(* PLC project MQTT, OpenPLC MQTT 1.0, author OpenPLC Lib Writter *)
(* stored: creationDateTime 2023-04-26T04:54:00, modificationDateTime 2023-04-26T04:54:00 *)

(* MQTT_RECEIVE *)
FUNCTION_BLOCK MQTT_RECEIVE
  VAR_INPUT
    RECEIVE : BOOL;  (* RECEIVE *)
    TOPIC : STRING;  (* TOPIC *)
  END_VAR
  VAR_OUTPUT
    RECEIVED : BOOL;  (* RECEIVED *)
    MESSAGE : STRING;  (* MESSAGE *)
  END_VAR

  RECEIVED := 0;
END_FUNCTION_BLOCK

(* MQTT_SEND *)
FUNCTION_BLOCK MQTT_SEND
  VAR_INPUT
    SEND : BOOL;  (* SEND *)
    TOPIC : STRING;  (* TOPIC *)
    MESSAGE : STRING;  (* MESSAGE *)
  END_VAR
  VAR_OUTPUT
    SUCCESS : BOOL;  (* SUCCESS *)
  END_VAR

  SUCCESS := 0;
END_FUNCTION_BLOCK

(* MQTT_CONNECT *)
FUNCTION_BLOCK MQTT_CONNECT
  VAR_INPUT
    CONNECT : BOOL;  (* CONNECT *)
    BROKER : STRING;  (* BROKER *)
    PORT : UINT;  (* PORT *)
  END_VAR
  VAR_OUTPUT
    SUCCESS : BOOL;  (* SUCCESS *)
  END_VAR

  SUCCESS := 0;
END_FUNCTION_BLOCK

(* MQTT_SUBSCRIBE *)
FUNCTION_BLOCK MQTT_SUBSCRIBE
  VAR_INPUT
    SUBSCRIBE : BOOL;  (* SUBSCRIBE *)
    TOPIC : STRING;  (* TOPIC *)
  END_VAR
  VAR_OUTPUT
    SUCCESS : BOOL;  (* SUCCESS *)
  END_VAR

  SUCCESS := 0;
END_FUNCTION_BLOCK
